ABB RobotStudio station: Solution1.rsstn

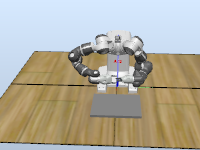
Station Solution1 (saved by RobotStudio 7.0.8746.631)
Controller IRB
  mechanical unit ROB_R: IRB14000_0.5_0.5_R, 6 joints, base frame (0, 0, 0) mm
  mechanical unit ROB_R_7: IRB14000_0.5_0.5_R, 1 joints, base frame (0, 0, 0) mm
  mechanical unit ROB_L: IRB14000_0.5_0.5_L, 6 joints, base frame (0, 0, 0) mm
  mechanical unit ROB_L_7: IRB14000_0.5_0.5_L, 1 joints, base frame (0, 0, 0) mm
Layout (positions relative to the parent item):
  - IRB14000_0.5_0.5 [mechanism, from Robots\IRB14000_0.5_0.5__01.rslib] at (0, 0, 0) mm
  - IRB14000_0.5_0.5_R [mechanism, from Robots\IRB14000_0.5_0.5__01.rslib] at (0, 0, 0) mm; joint values [1.1799, -1.4847, -1.4304, 0.6017, -0.4285, 0.7641, 0.9256] (rad or m)
  - IRB14000_0.5_0.5_L [mechanism, from Robots\IRB14000_0.5_0.5__01.rslib] at (0, 0, 0) mm; joint values [-1.4505, -2.3721, 0.9781, 0.7676, 1.347, 1.2563, -3.1944] (rad or m)
  - RightGripper [mechanism, from Tools\ABB_Smart_Gripper_Servo_Camera_Fingers.rslib] at (346.91, -135.98, 214.44) mm, rotated rx 71.48 ry -84.35 rz -161.36 deg; joint values [0.025] (rad or m)
  - LeftGripper [mechanism, from Tools\ABB_Smart_Gripper_Servo_Camera_Fingers.rslib] at (335.87, 124.46, 216.37) mm, rotated rx 89.1 ry -3.85 rz 6.43 deg; joint values [0.025] (rad or m)
  - floor [part]
  - table [part] at (0, -3.05, 0) mm
  - Cube [part] at (331.14, -19.91, 210.33) mm, rotated rx 30.43 ry 84.45 rz 31.4 deg
  - Integrated Vision camera Cam00X [part, from Equipment\IV_Cam00X.rslib] at (201.48, -2.61, 544.04) mm, rotated rx 179.29 ry 16.45 rz 177.01 deg
Attachment: RightGripper is attached to IRB14000_0.5_0.5_R / Link7
Attachment: LeftGripper is attached to IRB14000_0.5_0.5_L / Link7
EventTableEntry 1735: Group=, Trigger=DO_CloseGripper 1736, Actions=[EventTableActionMechanicalPose 1737, EventTableActionAttach 1745, EventTableActionDetach 2602], Comment=, ActivationMode=2, Cyclic=false
EventTableTriggerIO 1736: IOValue=[1], IRC5Controller=? -1, Operator=0, SignalSource=IRB 515
EventTableActionMechanicalPose 1737: VirtualSignal=SS_GripperIsClosed, Mechanism=RightGripper 1560, ToPoseName=PoseClose, VirtualSignalValue=[1]
EventTableEntry 1738: Group=, Trigger=DO_CloseGripper 1739, Actions=[EventTableActionMechanicalPose 1740, EventTableActionDetach 1747], Comment=, ActivationMode=2, Cyclic=false
EventTableTriggerIO 1739: IOValue=[0], IRC5Controller=? -1, Operator=0, SignalSource=IRB 515
EventTableActionMechanicalPose 1740: VirtualSignal=SS_GripperIsClosed, Mechanism=RightGripper 1560, ToPoseName=PoseOpen, VirtualSignalValue=[0]
EventTableEntry 1741: Group=, Trigger=NOP 1742, Actions=[DI_GripperIsClosed 1744], Comment=, ActivationMode=2, Cyclic=false
EventTableTriggerLogic 1742: layoutX=8, layoutY=16, Operand1=SS_GripperIsClosed 1743, Operand2=? -1, Operator=4, Delay=1000
EventTableTriggerIO 1743: IOValue=[-1], IRC5Controller=? -1, Operator=0, SignalSource=Solution1 1
EventTableActionIO 1744: IOValue=[-1], IRC5Controller=? -1, SignalTarget=IRB 515
EventTableActionAttach 1745: AttachmentParent=RightGripper 1560, AttachmentChild=Cube 1586, MountObject=false, Offset=[X=1, Y=0, Z=0, W=0, X=0, Y=1, Z=0, W=0, X=0, Y=0, Z=1, W=0, X=0, Y=0, Z=0, W=1], FlangeIndext=0, FindNearest=false
EventTableTriggerIO 1746: IOValue=[1], IRC5Controller=? -1, Operator=0, SignalSource=IRB 515
EventTableActionDetach 1747: AttachmentParent=RightGripper 1560, AttachmentChild=Cube 1586
EventTableTriggerIO 1748: IOValue=[0], IRC5Controller=? -1, Operator=0, SignalSource=IRB 515
EventTableTriggerLogic 1749: Operand1=SS_GripperIsClosed 1743, Operand2=? -1, Operator=4, Delay=1000
EventTableTriggerIO 1856: IOValue=[1], IRC5Controller=? -1, Operator=0, SignalSource=IRB 515
EventTableTriggerIO 1857: IOValue=[1], IRC5Controller=? -1, Operator=0, SignalSource=IRB 515
EventTableTriggerIO 1858: IOValue=[1], IRC5Controller=? -1, Operator=0, SignalSource=IRB 515
EventTableTriggerIO 1859: IOValue=[1], IRC5Controller=? -1, Operator=0, SignalSource=IRB 515
EventTableTriggerIO 1860: IOValue=[0], IRC5Controller=? -1, Operator=0, SignalSource=IRB 515
EventTableTriggerIO 1861: IOValue=[0], IRC5Controller=? -1, Operator=0, SignalSource=IRB 515
EventTableTriggerIO 1862: IOValue=[0], IRC5Controller=? -1, Operator=0, SignalSource=IRB 515
EventTableTriggerIO 1863: IOValue=[0], IRC5Controller=? -1, Operator=0, SignalSource=IRB 515
EventTableTriggerLogic 1864: layoutX=8, layoutY=16, Operand1=SS_GripperIsClosed 1743, Operand2=? -1, Operator=4, Delay=1000
EventTableTriggerLogic 1865: layoutX=8, layoutY=16, Operand1=SS_GripperIsClosed 1743, Operand2=? -1, Operator=4, Delay=1000
EventTableTriggerLogic 1866: layoutX=8, layoutY=16, Operand1=SS_GripperIsClosed 1743, Operand2=? -1, Operator=4, Delay=1000
EventTableTriggerLogic 1867: layoutX=8, layoutY=16, Operand1=SS_GripperIsClosed 1743, Operand2=? -1, Operator=4, Delay=1000
EventTableEntry 2089: Group=, Trigger=DO_CloseGripperL 2090, Actions=[EventTableActionMechanicalPose 2091, EventTableActionAttach 2130, EventTableActionDetach 2131], Comment=, ActivationMode=2, Cyclic=false
EventTableTriggerIO 2090: IOValue=[1], IRC5Controller=? -1, Operator=0, SignalSource=IRB 515
EventTableActionMechanicalPose 2091: VirtualSignal=SS_GripperIsClosedL, Mechanism=LeftGripper 1568, ToPoseName=PoseClose, VirtualSignalValue=[1]
EventTableEntry 2092: Group=, Trigger=DO_CloseGripperL 2093, Actions=[EventTableActionMechanicalPose 2094, EventTableActionDetach 2132], Comment=, ActivationMode=2, Cyclic=false
EventTableTriggerIO 2093: IOValue=[0], IRC5Controller=? -1, Operator=0, SignalSource=IRB 515
EventTableActionMechanicalPose 2094: VirtualSignal=SS_GripperIsClosedL, Mechanism=LeftGripper 1568, ToPoseName=PoseOpen, VirtualSignalValue=[0]
EventTableEntry 2095: Group=, Trigger=NOP 2096, Actions=[DI_GripperClosedL 2098], Comment=, ActivationMode=2, Cyclic=false
EventTableTriggerLogic 2096: Operand1=SS_GripperIsClosedL 2097, Operand2=? -1, Operator=4, Delay=1000
EventTableTriggerIO 2097: IOValue=[-1], IRC5Controller=? -1, Operator=0, SignalSource=Solution1 1
EventTableActionIO 2098: IOValue=[-1], IRC5Controller=? -1, SignalTarget=IRB 515
EventTableActionAttach 2130: AttachmentParent=LeftGripper 1568, AttachmentChild=Cube 1586, MountObject=false, Offset=[X=1, Y=0, Z=0, W=0, X=0, Y=1, Z=0, W=0, X=0, Y=0, Z=1, W=0, X=0, Y=0, Z=0, W=1], FlangeIndext=0, FindNearest=false
EventTableActionDetach 2131: AttachmentParent=RightGripper 1560, AttachmentChild=Cube 1586
EventTableActionDetach 2132: AttachmentParent=LeftGripper 1568, AttachmentChild=Cube 1586
EventTableTriggerIO 2448: IOValue=[1], IRC5Controller=? -1, Operator=0, SignalSource=IRB 515
EventTableTriggerIO 2449: IOValue=[1], IRC5Controller=? -1, Operator=0, SignalSource=IRB 515
EventTableTriggerIO 2450: IOValue=[1], IRC5Controller=? -1, Operator=0, SignalSource=IRB 515
EventTableTriggerIO 2451: IOValue=[1], IRC5Controller=? -1, Operator=0, SignalSource=IRB 515
EventTableTriggerIO 2452: IOValue=[0], IRC5Controller=? -1, Operator=0, SignalSource=IRB 515
EventTableTriggerIO 2453: IOValue=[0], IRC5Controller=? -1, Operator=0, SignalSource=IRB 515
EventTableTriggerIO 2454: IOValue=[0], IRC5Controller=? -1, Operator=0, SignalSource=IRB 515
EventTableTriggerIO 2455: IOValue=[0], IRC5Controller=? -1, Operator=0, SignalSource=IRB 515
EventTableTriggerLogic 2456: layoutX=8, layoutY=16, Operand1=SS_GripperIsClosed 1743, Operand2=? -1, Operator=4, Delay=1000
EventTableTriggerLogic 2457: layoutX=8, layoutY=16, Operand1=SS_GripperIsClosed 1743, Operand2=? -1, Operator=4, Delay=1000
EventTableTriggerLogic 2458: layoutX=8, layoutY=16, Operand1=SS_GripperIsClosed 1743, Operand2=? -1, Operator=4, Delay=1000
EventTableTriggerLogic 2459: layoutX=8, layoutY=16, Operand1=SS_GripperIsClosed 1743, Operand2=? -1, Operator=4, Delay=1000
EventTableTriggerIO 2460: IOValue=[1], IRC5Controller=? -1, Operator=0, SignalSource=IRB 515
EventTableTriggerIO 2461: IOValue=[1], IRC5Controller=? -1, Operator=0, SignalSource=IRB 515
EventTableTriggerIO 2462: IOValue=[1], IRC5Controller=? -1, Operator=0, SignalSource=IRB 515
EventTableTriggerIO 2463: IOValue=[1], IRC5Controller=? -1, Operator=0, SignalSource=IRB 515
EventTableTriggerIO 2464: IOValue=[0], IRC5Controller=? -1, Operator=0, SignalSource=IRB 515
EventTableTriggerIO 2465: IOValue=[0], IRC5Controller=? -1, Operator=0, SignalSource=IRB 515
EventTableTriggerIO 2466: IOValue=[0], IRC5Controller=? -1, Operator=0, SignalSource=IRB 515
EventTableTriggerIO 2467: IOValue=[0], IRC5Controller=? -1, Operator=0, SignalSource=IRB 515
EventTableTriggerLogic 2468: Operand1=SS_GripperIsClosedL 2097, Operand2=? -1, Operator=4, Delay=1000
EventTableTriggerLogic 2469: Operand1=SS_GripperIsClosedL 2097, Operand2=? -1, Operator=4, Delay=1000
EventTableTriggerLogic 2470: Operand1=SS_GripperIsClosedL 2097, Operand2=? -1, Operator=4, Delay=1000
EventTableTriggerLogic 2471: Operand1=SS_GripperIsClosedL 2097, Operand2=? -1, Operator=4, Delay=1000
EventTableEntry 2472: Group=, Trigger=NOP 2473, Actions=[DI_RightPermission 2475], Comment=, ActivationMode=2, Cyclic=false
EventTableTriggerLogic 2473: Operand1=DO_LeftAtPos 2474, Operand2=? -1, Operator=4, Delay=1000
EventTableTriggerIO 2474: IOValue=[-1], IRC5Controller=? -1, Operator=0, SignalSource=IRB 515
EventTableActionIO 2475: IOValue=[-1], IRC5Controller=? -1, SignalTarget=IRB 515
EventTableTriggerLogic 2476: Operand1=DO_LeftAtPos 2474, Operand2=? -1, Operator=4, Delay=1000
EventTableTriggerLogic 2477: Operand1=DO_LeftAtPos 2474, Operand2=? -1, Operator=4, Delay=1000
EventTableTriggerLogic 2478: Operand1=DO_LeftAtPos 2474, Operand2=? -1, Operator=4, Delay=1000
EventTableTriggerLogic 2479: Operand1=DO_LeftAtPos 2474, Operand2=? -1, Operator=4, Delay=1000
EventTableEntry 2480: Group=, Trigger=NOP 2481, Actions=[DI_LeftPermission 2483], Comment=, ActivationMode=2, Cyclic=false
EventTableTriggerLogic 2481: Operand1=DO_RightAtPos 2482, Operand2=? -1, Operator=4, Delay=1000
EventTableTriggerIO 2482: IOValue=[-1], IRC5Controller=? -1, Operator=0, SignalSource=IRB 515
EventTableActionIO 2483: IOValue=[-1], IRC5Controller=? -1, SignalTarget=IRB 515
EventTableTriggerLogic 2484: Operand1=DO_RightAtPos 2482, Operand2=? -1, Operator=4, Delay=1000
EventTableTriggerLogic 2485: Operand1=DO_RightAtPos 2482, Operand2=? -1, Operator=4, Delay=1000
EventTableTriggerLogic 2486: Operand1=DO_RightAtPos 2482, Operand2=? -1, Operator=4, Delay=1000
EventTableTriggerLogic 2487: Operand1=DO_RightAtPos 2482, Operand2=? -1, Operator=4, Delay=1000
EventTableActionDetach 2602: AttachmentParent=LeftGripper 1568, AttachmentChild=Cube 1586
EventTableTriggerIO 2774: IOValue=[1], IRC5Controller=? -1, Operator=0, SignalSource=IRB 515
EventTableTriggerIO 2775: IOValue=[1], IRC5Controller=? -1, Operator=0, SignalSource=IRB 515
EventTableTriggerIO 2776: IOValue=[1], IRC5Controller=? -1, Operator=0, SignalSource=IRB 515
EventTableTriggerIO 2777: IOValue=[1], IRC5Controller=? -1, Operator=0, SignalSource=IRB 515
EventTableTriggerIO 2778: IOValue=[0], IRC5Controller=? -1, Operator=0, SignalSource=IRB 515
EventTableTriggerIO 2779: IOValue=[0], IRC5Controller=? -1, Operator=0, SignalSource=IRB 515
EventTableTriggerIO 2780: IOValue=[0], IRC5Controller=? -1, Operator=0, SignalSource=IRB 515
EventTableTriggerIO 2781: IOValue=[0], IRC5Controller=? -1, Operator=0, SignalSource=IRB 515
EventTableTriggerLogic 2782: layoutX=8, layoutY=16, Operand1=SS_GripperIsClosed 1743, Operand2=? -1, Operator=4, Delay=1000
EventTableTriggerLogic 2783: layoutX=8, layoutY=16, Operand1=SS_GripperIsClosed 1743, Operand2=? -1, Operator=4, Delay=1000
EventTableTriggerLogic 2784: layoutX=8, layoutY=16, Operand1=SS_GripperIsClosed 1743, Operand2=? -1, Operator=4, Delay=1000
EventTableTriggerLogic 2785: layoutX=8, layoutY=16, Operand1=SS_GripperIsClosed 1743, Operand2=? -1, Operator=4, Delay=1000
EventTableTriggerIO 2786: IOValue=[1], IRC5Controller=? -1, Operator=0, SignalSource=IRB 515
EventTableTriggerIO 2787: IOValue=[1], IRC5Controller=? -1, Operator=0, SignalSource=IRB 515
EventTableTriggerIO 2788: IOValue=[1], IRC5Controller=? -1, Operator=0, SignalSource=IRB 515
EventTableTriggerIO 2789: IOValue=[1], IRC5Controller=? -1, Operator=0, SignalSource=IRB 515
EventTableTriggerIO 2790: IOValue=[0], IRC5Controller=? -1, Operator=0, SignalSource=IRB 515
EventTableTriggerIO 2791: IOValue=[0], IRC5Controller=? -1, Operator=0, SignalSource=IRB 515
EventTableTriggerIO 2792: IOValue=[0], IRC5Controller=? -1, Operator=0, SignalSource=IRB 515
EventTableTriggerIO 2793: IOValue=[0], IRC5Controller=? -1, Operator=0, SignalSource=IRB 515
EventTableTriggerLogic 2794: Operand1=SS_GripperIsClosedL 2097, Operand2=? -1, Operator=4, Delay=1000
EventTableTriggerLogic 2795: Operand1=SS_GripperIsClosedL 2097, Operand2=? -1, Operator=4, Delay=1000
EventTableTriggerLogic 2796: Operand1=SS_GripperIsClosedL 2097, Operand2=? -1, Operator=4, Delay=1000
EventTableTriggerLogic 2797: Operand1=SS_GripperIsClosedL 2097, Operand2=? -1, Operator=4, Delay=1000
EventTableTriggerLogic 2798: Operand1=DO_LeftAtPos 2474, Operand2=? -1, Operator=4, Delay=1000
EventTableTriggerLogic 2799: Operand1=DO_LeftAtPos 2474, Operand2=? -1, Operator=4, Delay=1000
EventTableTriggerLogic 2800: Operand1=DO_LeftAtPos 2474, Operand2=? -1, Operator=4, Delay=1000
EventTableTriggerLogic 2801: Operand1=DO_LeftAtPos 2474, Operand2=? -1, Operator=4, Delay=1000
EventTableTriggerLogic 2802: Operand1=DO_RightAtPos 2482, Operand2=? -1, Operator=4, Delay=1000
EventTableTriggerLogic 2803: Operand1=DO_RightAtPos 2482, Operand2=? -1, Operator=4, Delay=1000
EventTableTriggerLogic 2804: Operand1=DO_RightAtPos 2482, Operand2=? -1, Operator=4, Delay=1000
EventTableTriggerLogic 2805: Operand1=DO_RightAtPos 2482, Operand2=? -1, Operator=4, Delay=1000
EventTableTriggerIO 2942: IOValue=[1], IRC5Controller=? -1, Operator=0, SignalSource=IRB 515
EventTableTriggerIO 2943: IOValue=[1], IRC5Controller=? -1, Operator=0, SignalSource=IRB 515
EventTableTriggerIO 2944: IOValue=[0], IRC5Controller=? -1, Operator=0, SignalSource=IRB 515
EventTableTriggerIO 2945: IOValue=[0], IRC5Controller=? -1, Operator=0, SignalSource=IRB 515
EventTableTriggerLogic 2946: layoutX=8, layoutY=16, Operand1=SS_GripperIsClosed 1743, Operand2=? -1, Operator=4, Delay=1000
EventTableTriggerLogic 2947: layoutX=8, layoutY=16, Operand1=SS_GripperIsClosed 1743, Operand2=? -1, Operator=4, Delay=1000
EventTableTriggerIO 2948: IOValue=[1], IRC5Controller=? -1, Operator=0, SignalSource=IRB 515
EventTableTriggerIO 2949: IOValue=[1], IRC5Controller=? -1, Operator=0, SignalSource=IRB 515
EventTableTriggerIO 2950: IOValue=[0], IRC5Controller=? -1, Operator=0, SignalSource=IRB 515
EventTableTriggerIO 2951: IOValue=[0], IRC5Controller=? -1, Operator=0, SignalSource=IRB 515
EventTableTriggerLogic 2952: Operand1=SS_GripperIsClosedL 2097, Operand2=? -1, Operator=4, Delay=1000
EventTableTriggerLogic 2953: Operand1=SS_GripperIsClosedL 2097, Operand2=? -1, Operator=4, Delay=1000
EventTableTriggerLogic 2954: Operand1=DO_LeftAtPos 2474, Operand2=? -1, Operator=4, Delay=1000
EventTableTriggerLogic 2955: Operand1=DO_LeftAtPos 2474, Operand2=? -1, Operator=4, Delay=1000
EventTableTriggerLogic 2956: Operand1=DO_RightAtPos 2482, Operand2=? -1, Operator=4, Delay=1000
EventTableTriggerLogic 2957: Operand1=DO_RightAtPos 2482, Operand2=? -1, Operator=4, Delay=1000
EventTableTriggerIO 2964: IOValue=[1], IRC5Controller=? -1, Operator=0, SignalSource=IRB 515
EventTableTriggerIO 2965: IOValue=[1], IRC5Controller=? -1, Operator=0, SignalSource=IRB 515
EventTableTriggerIO 2966: IOValue=[1], IRC5Controller=? -1, Operator=0, SignalSource=IRB 515
EventTableTriggerIO 2967: IOValue=[1], IRC5Controller=? -1, Operator=0, SignalSource=IRB 515
EventTableTriggerIO 2968: IOValue=[1], IRC5Controller=? -1, Operator=0, SignalSource=IRB 515
EventTableTriggerIO 2969: IOValue=[0], IRC5Controller=? -1, Operator=0, SignalSource=IRB 515
EventTableTriggerIO 2970: IOValue=[0], IRC5Controller=? -1, Operator=0, SignalSource=IRB 515
EventTableTriggerIO 2971: IOValue=[0], IRC5Controller=? -1, Operator=0, SignalSource=IRB 515
EventTableTriggerIO 2972: IOValue=[0], IRC5Controller=? -1, Operator=0, SignalSource=IRB 515
EventTableTriggerIO 2973: IOValue=[0], IRC5Controller=? -1, Operator=0, SignalSource=IRB 515
EventTableTriggerLogic 2974: layoutX=8, layoutY=16, Operand1=SS_GripperIsClosed 1743, Operand2=? -1, Operator=4, Delay=1000
EventTableTriggerLogic 2975: layoutX=8, layoutY=16, Operand1=SS_GripperIsClosed 1743, Operand2=? -1, Operator=4, Delay=1000
EventTableTriggerLogic 2976: layoutX=8, layoutY=16, Operand1=SS_GripperIsClosed 1743, Operand2=? -1, Operator=4, Delay=1000
EventTableTriggerLogic 2977: layoutX=8, layoutY=16, Operand1=SS_GripperIsClosed 1743, Operand2=? -1, Operator=4, Delay=1000
EventTableTriggerLogic 2978: layoutX=8, layoutY=16, Operand1=SS_GripperIsClosed 1743, Operand2=? -1, Operator=4, Delay=1000
EventTableTriggerIO 2979: IOValue=[1], IRC5Controller=? -1, Operator=0, SignalSource=IRB 515
EventTableTriggerIO 2980: IOValue=[1], IRC5Controller=? -1, Operator=0, SignalSource=IRB 515
EventTableTriggerIO 2981: IOValue=[1], IRC5Controller=? -1, Operator=0, SignalSource=IRB 515
EventTableTriggerIO 2982: IOValue=[1], IRC5Controller=? -1, Operator=0, SignalSource=IRB 515
EventTableTriggerIO 2983: IOValue=[1], IRC5Controller=? -1, Operator=0, SignalSource=IRB 515
EventTableTriggerIO 2984: IOValue=[0], IRC5Controller=? -1, Operator=0, SignalSource=IRB 515
EventTableTriggerIO 2985: IOValue=[0], IRC5Controller=? -1, Operator=0, SignalSource=IRB 515
EventTableTriggerIO 2986: IOValue=[0], IRC5Controller=? -1, Operator=0, SignalSource=IRB 515
EventTableTriggerIO 2987: IOValue=[0], IRC5Controller=? -1, Operator=0, SignalSource=IRB 515
EventTableTriggerIO 2988: IOValue=[0], IRC5Controller=? -1, Operator=0, SignalSource=IRB 515
EventTableTriggerLogic 2989: Operand1=SS_GripperIsClosedL 2097, Operand2=? -1, Operator=4, Delay=1000
EventTableTriggerLogic 2990: Operand1=SS_GripperIsClosedL 2097, Operand2=? -1, Operator=4, Delay=1000
EventTableTriggerLogic 2991: Operand1=SS_GripperIsClosedL 2097, Operand2=? -1, Operator=4, Delay=1000
EventTableTriggerLogic 2992: Operand1=SS_GripperIsClosedL 2097, Operand2=? -1, Operator=4, Delay=1000
EventTableTriggerLogic 2993: Operand1=SS_GripperIsClosedL 2097, Operand2=? -1, Operator=4, Delay=1000
EventTableTriggerLogic 2994: Operand1=DO_LeftAtPos 2474, Operand2=? -1, Operator=4, Delay=1000
EventTableTriggerLogic 2995: Operand1=DO_LeftAtPos 2474, Operand2=? -1, Operator=4, Delay=1000
EventTableTriggerLogic 2996: Operand1=DO_LeftAtPos 2474, Operand2=? -1, Operator=4, Delay=1000
EventTableTriggerLogic 2997: Operand1=DO_LeftAtPos 2474, Operand2=? -1, Operator=4, Delay=1000
EventTableTriggerLogic 2998: Operand1=DO_LeftAtPos 2474, Operand2=? -1, Operator=4, Delay=1000
EventTableTriggerLogic 2999: Operand1=DO_RightAtPos 2482, Operand2=? -1, Operator=4, Delay=1000
EventTableTriggerLogic 3000: Operand1=DO_RightAtPos 2482, Operand2=? -1, Operator=4, Delay=1000
EventTableTriggerLogic 3001: Operand1=DO_RightAtPos 2482, Operand2=? -1, Operator=4, Delay=1000
EventTableTriggerLogic 3002: Operand1=DO_RightAtPos 2482, Operand2=? -1, Operator=4, Delay=1000
EventTableTriggerLogic 3003: Operand1=DO_RightAtPos 2482, Operand2=? -1, Operator=4, Delay=1000
Station signals: DI SS_GripperIsClosed, DI SS_GripperIsClosedL
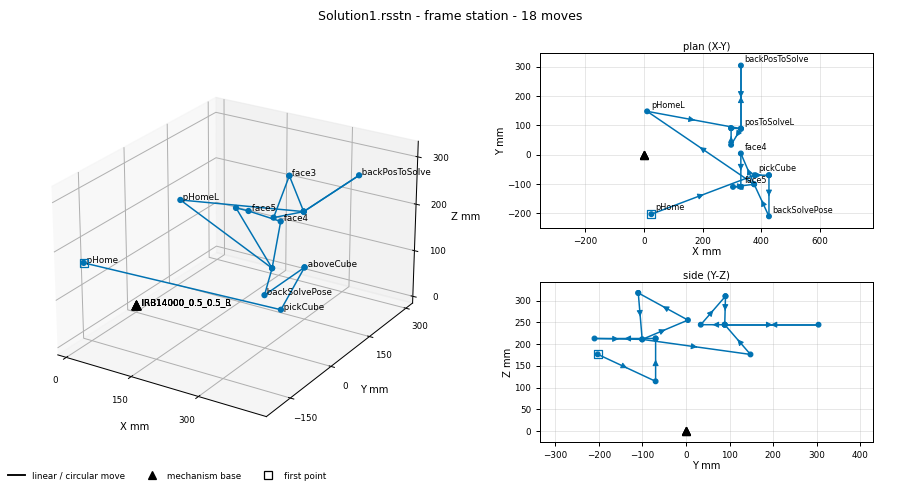
[picture p0: tool path of Solution1.rsstn in frame station, 18 of 18 moves have a stored position in this frame; points joined in program order, loops and branches not executed]
Targets, tools, work objects and paths stored in the station, written as RAPID:
! task T_ROB_R
MODULE CalibData
  PERS tooldata Servo:=[TRUE,[[0,0,114.2],[1,0,0,0]],[0.229,[7.9,12.4,48.7],[1,0,0,0],0.00021,0.00023,0.00008]];
  PERS tooldata Camera:=[TRUE,[[-7.3,28.3,35.1],[0.5,-0.5,0.5,0.5]],[0.229,[7.9,12.4,48.7],[1,0,0,0],0.00021,0.00023,0.00008]];
  TASK PERS wobjdata Workobject_2:=[FALSE,TRUE,"",[[0,0,0],[1,0,0,0]],[[0,0,0],[1,0,0,0]]];
  TASK PERS wobjdata Workobject_3:=[FALSE,TRUE,"",[[0,0,0],[1,0,0,0]],[[0,0,0],[1,0,0,0]]];
ENDMODULE

! task T_ROB_R
MODULE Module1
  CONST robtarget pHome:=[[24.971763923,-202.839465162,176.64502516],[0.07106331,0.248288947,-0.660142697,0.705346883],[0,0,0,4],[-101.964427132,9E+09,9E+09,9E+09,9E+09,9E+09]];
  CONST robtarget pickCube:=[[376.766775496,-69.805089288,114.555214565],[0.693258996,-0.185986842,-0.178114343,-0.673109307],[1,-1,0,4],[-118.392955921,9E+09,9E+09,9E+09,9E+09,9E+09]];
  CONST robtarget aboveCube:=[[426.254207357,-69.807230037,212.96301894],[0.648575132,-0.580206927,0.34163322,-0.35496051],[1,0,1,4],[-162.757998243,9E+09,9E+09,9E+09,9E+09,9E+09]];
  CONST robtarget posToSolve:=[[426.254207357,-69.807230037,212.96301894],[0.648575132,-0.580206927,0.34163322,-0.35496051],[1,0,1,4],[-162.757998243,9E+09,9E+09,9E+09,9E+09,9E+09]];
  CONST robtarget posToSolveL:=[[330.258737132,106.2649604,244.629751284],[0.667938754,-0.028125826,-0.019909493,0.743418033],[-1,1,-2,4],[106.437394206,9E+09,9E+09,9E+09,9E+09,9E+09]];
  CONST robtarget pHomeL:=[[10.457496534,148.132867885,176.35475559],[0.248288947,0.07106331,-0.705346883,0.660142697],[0,0,0,4],[101.964427132,9E+09,9E+09,9E+09,9E+09,9E+09]];
  CONST robtarget backSolvePose:=[[426.254927622,-210.235279713,212.962526197],[0.64857477,-0.580207492,0.341633336,-0.354960135],[1,0,1,4],[-162.757997875,9E+09,9E+09,9E+09,9E+09,9E+09]];
  CONST robtarget posToSolve2:=[[375.645423458,-100.654462746,210.914642182],[0.53109775,-0.468723047,0.483378506,-0.514372535],[1,0,1,4],[-162.757996376,9E+09,9E+09,9E+09,9E+09,9E+09]];
  CONST robtarget face4:=[[330.361100068,4.444400586,255.255095174],[0.832317803,0.039463524,0.552341666,-0.024665535],[1,0,0,4],[-162.68678863,9E+09,9E+09,9E+09,9E+09,9E+09]];
  CONST robtarget face5:=[[330.362428827,-109.679264893,317.635430954],[0.736460496,0.167175431,-0.113108623,-0.645666131],[1,0,0,4],[-162.686785121,9E+09,9E+09,9E+09,9E+09,9E+09]];
  CONST robtarget face6:=[[303.58293492,-109.680765697,317.634844572],[0.129110416,-0.641874856,0.733824267,-0.181188063],[1,0,-2,4],[-162.686786056,9E+09,9E+09,9E+09,9E+09,9E+09]];
  PROC main()
    MoveL pHome,v300,z100,Camera\WObj:=wobj0;
    MoveL pickCube,v300,fine,Camera\WObj:=Workobject_2;
    SetDO DO_CloseGripper,1;
    WaitDI DI_GripperIsClosed,1;
    MoveL aboveCube,v300,fine,Camera\WObj:=Workobject_2;
    MoveL posToSolve,v300,fine,Camera\WObj:=Workobject_2;
    SetDO DO_RightAtPos,1;
    WaitDI DI_RightPermission,1;
    SetDO DO_CloseGripper,0;
    WaitDI DI_GripperIsClosed,0;
    MoveL backSolvePose,v300,fine,Camera\WObj:=Workobject_2;
    SetDO DO_RightAtPos,0;
    WaitDI DI_RightPermission,0;
    MoveL posToSolve2,v300,fine,Camera\WObj:=Workobject_2;
    SetDO DO_CloseGripper,1;
    WaitDI DI_GripperIsClosed,1;
    SetDO DO_RightAtPos,1;
    WaitDI DI_RightPermission,1;
    MoveL face4,v80,fine,Camera\WObj:=Workobject_2;
    MoveL face5,v100,fine,Camera\WObj:=Workobject_2;
    MoveL face6,v30,fine,Camera\WObj:=Workobject_2;
    MoveL posToSolve2,v80,fine,Camera\WObj:=Workobject_2;
    SetDO DO_RightAtPos,0;
  ENDPROC
ENDMODULE

! task T_ROB_L
MODULE CalibData
  PERS tooldata Servo:=[TRUE,[[0,0,114.2],[1,0,0,0]],[0.229,[7.9,12.4,48.7],[1,0,0,0],0.00021,0.00023,0.00008]];
  PERS tooldata Camera:=[TRUE,[[-7.3,28.3,35.1],[0.5,-0.5,0.5,0.5]],[0.229,[7.9,12.4,48.7],[1,0,0,0],0.00021,0.00023,0.00008]];
  TASK PERS wobjdata Workobject_3:=[FALSE,TRUE,"",[[0,0,0],[1,0,0,0]],[[0,0,0],[1,0,0,0]]];
ENDMODULE

! task T_ROB_L
MODULE Module1
  CONST robtarget pHomeL:=[[10.457496534,148.132867885,176.35475559],[0.248288947,0.07106331,-0.705346883,0.660142697],[0,0,0,4],[101.964427132,9E+09,9E+09,9E+09,9E+09,9E+09]];
  CONST robtarget posToSolveL:=[[330.588726687,88.996694067,244.663346065],[0.666138699,-0.028237347,-0.019784056,0.745030521],[-1,1,-2,4],[106.437512435,9E+09,9E+09,9E+09,9E+09,9E+09]];
  CONST robtarget face1:=[[297.108765245,33.934637119,244.662410778],[0.535895442,-0.568456493,0.421408825,0.460530013],[-1,0,-2,4],[106.437553404,9E+09,9E+09,9E+09,9E+09,9E+09]];
  CONST robtarget face2:=[[297.109440488,90.733841,310.176728249],[0.771903759,-0.111646776,-0.117222446,0.614783281],[-1,1,-2,4],[106.437564975,9E+09,9E+09,9E+09,9E+09,9E+09]];
  CONST robtarget face3:=[[297.10981702,90.73431925,310.176563128],[0.217827049,0.59473309,0.749751947,0.191614055],[0,-1,-3,4],[-159.430070068,9E+09,9E+09,9E+09,9E+09,9E+09]];
  CONST robtarget backPosToSolve:=[[330.589050351,304.441694714,244.663279056],[0.666138818,-0.028237032,-0.019784093,0.745030426],[-1,1,-2,4],[106.437510753,9E+09,9E+09,9E+09,9E+09,9E+09]];
  PROC main()
    MoveL pHomeL,v300,z100,Camera\WObj:=wobj0;
    WaitDI DI_LeftPermission,1;
    MoveL posToSolveL,v300,fine,Camera\WObj:=Workobject_3;
    SetDO DO_CloseGripperL,1;
    WaitDO DO_CloseGripperL,1;
    SetDO DO_LeftAtPos,1;
    WaitDI DI_LeftPermission,0;
    MoveL face1,v60,fine,Camera\WObj:=Workobject_3;
    MoveL face3,v60,fine,Camera\WObj:=Workobject_3;
    MoveL face2,v60,fine,Camera\WObj:=Workobject_3;
    MoveL posToSolveL,v100,fine,Camera\WObj:=Workobject_3;
    SetDO DO_LeftATPos,0;
    WaitDI DI_LeftPermission,1;
    SetDO DO_CloseGripperL,0;
    WaitDO DO_CloseGripperL,0;
    MoveL backPosToSolve,v300,fine,Camera\WObj:=Workobject_3;
    SetDO DO_LeftATPos,1;
    WaitDI DI_LeftPermission,0;
    MoveL posToSolveL,v300,fine,Camera\WObj:=Workobject_3;
  ENDPROC
ENDMODULE

